FUNCTION_BLOCK RobotControlSystem
VAR_INPUT
	Enable: BOOL;
	mxABBMoveStart: BOOL;
	mwTargetX: INT;
	mwTargetY: INT;
END_VAR
VAR_OUTPUT
END_VAR
VAR
	ABBMove: INT;
	RSpeed:INT:=1;
END_VAR

VAR_IN_OUT
	mwRobotXaxis: INT;
	mwRobotYaxis: INT;
END_VAR

IF Enable THEN
	CASE ABBMove OF
		0:
			IF mxABBMoveStart THEN
				ABBMove:=10;
			END_IF
		10:
			IF NOT CommData.mxABBExecuting THEN
				CommData.mxABBExecuting:=TRUE;
				ABBMove:=20;
			END_IF
		20:
			IF mwRobotXaxis < mwTargetX THEN
				mwRobotXaxis :=mwRobotXaxis+RSpeed;
				ABBMove:=30;
			ELSIF mwRobotXaxis > mwTargetX THEN
				mwRobotXaxis :=mwRobotXaxis-RSpeed;
				ABBMove:=30;
			ELSIF mwRobotXaxis = mwTargetX THEN
				ABBMove:=30;
			END_IF
		30:
			IF mwRobotYaxis < mwTargetY THEN
				mwRobotYaxis :=mwRobotYaxis+RSpeed;
				ABBMove:=40;
			ELSIF mwRobotYaxis > mwTargetY THEN
				mwRobotYaxis :=mwRobotYaxis-RSpeed;
				ABBMove:=40;
			ELSIF mwRobotYaxis = mwTargetY THEN
				ABBMove:=40;
			END_IF
		40:
			IF mwRobotXaxis = mwTargetX AND mwRobotYaxis = mwTargetY THEN
				ABBMove:=50;
			ELSIF gvl.ixEmergencyStop THEN
				ABBMove:=50;
			ELSE
				ABBMOve:=20;
			END_IF
		50:
			CommData.mxABBExecuting:=FALSE;
			IF NOT mxABBMoveStart THEN
				ABBMove:=0;
			END_IF
	END_CASE
END_IF

END_FUNCTION_BLOCK

(* stored: Version 1.1.0.1, ProductVersion 3.1.4024.12
   POU RobotControlSystem: Id {f6e2fbe6-3561-4b9f-9545-d178090ca923}, SpecialFunc None *)
